// TIA Portal V21 export
TYPE "Rcp_DataIn_Type"
   STRUCT
      Rcp_Edit : Int;   // index - editing recipe
      Rcp_Work : Int;   // index - actual recipe
      Rcp_Dest : Int;   // index - destination of copy
      Enable_changeover_condition : Array[0..9] of Bool;   // condizioni singole per abilitazione cambio ricetta (in popup)
      Enable_Changeover : Bool;   // enable "Load_in_Work" function
   END_STRUCT;
END_TYPE
